INTERFACE I_ServerResponseHeader

METHOD PUBLIC ToString
VAR_INPUT
	Destination : REFERENCE TO STRING(Constants.RESPONSE_HEADER_STRING_SIZE);
END_VAR
END_METHOD

METHOD PUBLIC TryGetField : BOOL;
VAR_INPUT
	Key : STRING;
	Destination : ANY;
END_VAR
END_METHOD

METHOD PUBLIC TryWriteField : BOOL;
VAR_INPUT
	Key : STRING;
	Source : ANY;
END_VAR
END_METHOD

END_INTERFACE

(* stored: Version 1.1.0.1, ProductVersion 3.1.4024.12
   Itf I_ServerResponseHeader: Id {c6e1f27a-5582-4ccb-bee1-25638f811636}
   Method ToString: Id {87083345-4611-4dde-93e5-ca9bbb47ae82}
   Method TryGetField: Id {fe6fd5d1-3b7c-4375-8f49-aead63fa0dd6}
   Method TryWriteField: Id {fbd1a505-b230-41e8-99d5-a5addaeeeff0} *)
